{attribute 'no_check'}
FUNCTION_BLOCK Cylinder_wUnitItf EXTENDS cylinder
VAR_OUTPUT CONSTANT
{attribute 'displaymode':='binary'}
	OPTION_REPORT_ERROR										:	BYTE := 2#0000_0001; //Set master unit into error if acuator is in error	
END_VAR
VAR_INPUT  
VAR_OUTPUT CONSTANT
{attribute 'displaymode':='binary'}
	Options													:	BYTE :=0;	
	ipUnit													:	I_StatemodelBase;	
	
END_VAR                                     			
VAR_OUTPUT 
	BtnBasePos												:	BOOL;		
	BtnWorkPos												:	BOOL;         			
END_VAR
VAR
END_VAR

	(* 										 								       	*)
	(* 								 												*)
	(********************************************************************************)

(* execute cylinder function *************************************)
	SUPER^();
	
(* Check master unit ***********************************************)
	IF ipUnit <> 0 
	THEN
		CASE ipUnit.actState OF
 		eSTATE.EXECUTE:
			IF ipUnit.actMode = eMODE.MANUAL OR ipUnit.mode = eMODE.SERVICE
			THEN
				IF BtnBasePos THEN SUPER^.moveToBasePos(); END_IF
				ELSIF BtnWorkPos THEN SUPER^.moveToWorkPos(); END_IF
			ELSE //In auto
				IF Options.0 AND_THEN SUPER^.inError
				THEN
					ipUnit.setMachineError();
				END_IF	
			END_IF
		END_CASE
	END_IF
	
(*********************************************************************)

END_FUNCTION_BLOCK

(* stored: Version 1.1.0.1, ProductVersion 3.1.4024.3
   POU Cylinder_wUnitItf: Id {0ab8f445-21f2-424b-be28-b865cad33352}, SpecialFunc None *)
